PROGRAM Controls
VAR
	MainState	:	INT;// 0 : OFF || 1 : manual Mode | 2 : AutoMode
END_VAR


IF Blower.OnPushBTN AND Blower.AutoPushBTN = FALSE AND Blower.AutoPushBTN = FALSE AND MainState <> 2 THEN
	
	MainState				:=	1;
	
END_IF

IF Blower.OffPushBTN THEN
	
	Mainstate				:=	0;
	Blower.AirBlowerPower	:=	FALSE;
	Blower.AutoPushBTN		:=	FALSE;
	Blower.OnPushBTN		:=	FALSE;
	
END_IF

IF Blower.AutoPushBTN AND Blower.OffPushBTN = FALSE AND Blower.OnPushBTN = FALSE THEN
	
	MainState 				:=	2;
	
END_IF

IF (Blower.OnPushBTN OR Blower.AutoPushBTN) AND Blower.OffPushBTN = FALSE  THEN
	
	Blower.AirBlowerPower	:=	TRUE;
	
END_IF

END_PROGRAM

(* stored: Version 1.1.0.1, ProductVersion 3.1.4024.9
   POU Controls: Id {134dc9d1-6b4a-4fde-8d27-9060ec6338ea}, SpecialFunc None *)
